FUNCTION Convert_USINT_TO_BOOL : BOOL
VAR_INPUT
	in : USINT;
	out : REFERENCE TO BOOL;
END_VAR
VAR
	converted : BOOL;
END_VAR

converted := USINT_TO_BOOL(in);

IF (BOOL_TO_USINT(converted) <> in) THEN
	RETURN;
END_IF

out := converted;
Convert_USINT_TO_BOOL := TRUE;

END_FUNCTION

(* stored: Version 1.1.0.1, ProductVersion 3.1.4024.12
   POU Convert_USINT_TO_BOOL: Id {7ea4887c-9ba7-46c1-a4c3-a1db4d46dcbe}, SpecialFunc None *)
